// TIA Portal V17 export
// export: Created 2025-03-10T12:18:14.0591614Z, ExportSetting WithDefaults, DisplayName Totally Integrated Automation Portal, DisplayVersion V17 Update 8, DisplayName TIA Portal Openness, DisplayVersion V17 Update 8, DisplayName TIA Portal Version Control Interface, DisplayVersion V17, DisplayName SINAMICS Startdrive Advanced, DisplayVersion V17 SP2, DisplayName SINAMICS Startdrive G110M, G120, G120C, G120D, G120P, G115D, DisplayVersion V17 SP2, DisplayName SINAMICS Startdrive G130, G150, S120, S150, SINAMICS MV, S210, DisplayVersion V17 SP2, DisplayName STEP 7 Professional, DisplayVersion V17 Update 8, DisplayName SINUMERIK ONE STEP 7 Toolbox, DisplayVersion V17 Update 12, DisplayName SINUMERIK 840D sl STEP 7 Toolbox, DisplayVersion V17 Update 12, DisplayName STEP 7 Safety, DisplayVersion V17 Update 6, DisplayName WinCC Advanced, DisplayVersion V17 Update 8
TYPE "HMI_SERVICE"
// stored: IsFailsafeCompliant false
   STRUCT
      HMI_START : Bool;
      HMI_STOP : Bool;
      HMI_STARTING : Bool;
      HMI_STOPPING : Bool;
      HMI_STARTED : Bool;
      HMI_STOPPED : Bool;
      HMI_START_CONDITIONS : Bool;
      HMI_STOP_CONDITIONS : Bool;
      FAULTED : Bool;
   END_STRUCT;
END_TYPE
